FUNCTION_BLOCK FB_CoolingNetwork
VAR_INPUT
	//control struct for cn
	controlAutomatic : ST_CoolingNetworkControl;	
END_VAR
VAR_OUTPUT
	{attribute 'OPC.UA.DA' := '1'}
	localState : ST_ThermalNetworkState;
END_VAR
VAR
	//systems
	BufferStorage : FB_BufferStorage;
	eChillerSystem : FB_eChillerSystem;
	HVFASystem : FB_HVFAStorageSystem;
	CentralMachineCoolingSystem : FB_CN_CentralMachineCooling;
	FlywheelMassStorageSystem : FB_FlywheelMassStorageSystem;
	
	//machines
	EMAG_GT : FB_EMAG_GT;
	FlyhweelMassStorage : FB_FlywheelMassStorage;
	
	//internal variables
	bSetStatusOn_CentralMachineCooling : BOOL;
	bSetStatusOn_FlywheelMassStorage : BOOL;
END_VAR

//buffer storage system
BufferStorage();
localState.fUpperTemperature := BufferStorage.localState.fUpperTemperature;
localState.fMidTemperature := BufferStorage.localState.fMidTemperature;
localState.fLowerTemperature := BufferStorage.localState.fLowerTemperature;
localState.fUpperTemperature_ActiveStorage := HVFASystem.localState.fUpperTemperature;
localState.fLowerTemperature_ActiveStorage := HVFASystem.localState.fLowerTemperature;

//machines
EMAG_GT();
bSetStatusOn_CentralMachineCooling := EMAG_GT.bStatusOn;
FlyhweelMassStorage();
bSetStatusOn_FlywheelMassStorage := FlyhweelMassStorage.bStatusOn;

//producer
eChillerSystem(bSetStatusOnAutomatic := controlAutomatic.bSetStatusOn_eChiller,
	bAlgorithmPermission := controlAutomatic.bAlgorithmPermission,
	fSetPointAutomatic := controlAutomatic.fFeedTemperature,
	fExternalTemperature := BufferStorage.localState.fMidTemperature,
	fReturnTemperature_Consumers := BufferStorage.localState.fUpperTemperature);

//consumer
//PU100 in central machine cooling system controls return temperature of 20 degree
CentralMachineCoolingSystem(bSetStatusOnAutomatic := bSetStatusOn_CentralMachineCooling,
	bAlgorithmPermission := controlAutomatic.bAlgorithmPermission,
	fSetPointAutomatic := 20);

//PU191 in central machine cooling system controls return temperature of 20 degree
FlywheelMassStorageSystem(bSetStatusOnAutomatic := bSetStatusOn_FlywheelMassStorage,
	bAlgorithmPermission := controlAutomatic.bAlgorithmPermission,
	fSetPointAutomatic := 20);
	
//external storages
HVFASystem(bSetStatusOnAutomatic := controlAutomatic.bSetStatusOn_HVFASystem,
	bAlgorithmPermission := controlAutomatic.bAlgorithmPermission,
	fSetPointAutomatic := 40,
	bLoadingAutomatic := controlAutomatic.bLoading_HVFASystem,
	aTelegramm_WMZ7x0 := aTelegramm_WMZ710,
	aTelegramm_WMZx05 := aTelegramm_WMZ105);

END_FUNCTION_BLOCK

(* stored: Version 1.1.0.1, ProductVersion 3.1.4024.10
   POU FB_CoolingNetwork: Id {3e3c7edc-aa3e-40d5-adb7-105c87a52325}, SpecialFunc None *)
